FUNCTION_BLOCK FB_FieldCodecUInt32 IMPLEMENTS I_FieldCodec
VAR_INPUT
END_VAR
VAR_OUTPUT
END_VAR
VAR
    nValue : DINT;
END_VAR

METHOD CalculatePackedDataSize : HRESULT
VAR_INPUT CONSTANT
	anyFirstElem	: T_Any;
	nLength	        : UDINT;        // items to write
END_VAR
VAR_OUTPUT
    nPackedDataSize : UDINT;
END_VAR
VAR
    anyItem         : T_ANY;
    i               : UDINT;
    nValue          : UDINT;
END_VAR
anyItem := anyFirstElem;

IF nLength < 1 THEN
    nPackedDataSize := 0;
    RETURN;
END_IF

FOR i := 0  TO nLength - 1 DO
    anyItem.pValue := anyFirstElem.pValue + (i * TO_UDINT(anyFirstElem.diSize));
    MEMCPY(destAddr:= ADR(nValue), srcAddr:= anyItem.pValue, n:= TO_UDINT(anyFirstElem.diSize));
    nPackedDataSize := nPackedDataSize + F_ComputeUInt32Size(nValue);
END_FOR
END_METHOD

METHOD IsPackedRepeatedField : BOOL
VAR_INPUT
	nTag	: UDINT;
END_VAR
IsPackedRepeatedField := F_IsPackedRepeatedField(nTag);
END_METHOD


METHOD ValueReader : HRESULT
VAR_IN_OUT      
    stCtx : ST_ParseContext;
END_VAR
VAR_OUTPUT
	anyOut	: T_Any;
END_VAR

ValueReader := F_ParseRawVarint32(stCtx, nValue);
anyOut := F_ToAnyType(anyArg:= nValue);
END_METHOD

METHOD ValueWriter : HRESULT
VAR_IN_OUT
    stCtx  : ST_WriteContext;
END_VAR
VAR_INPUT
	anyIn	: ANY;
END_VAR
VAR
    nValue  : UDINT;
END_VAR

// nValue := PUDINT_TO_UDINT(anyIn.pValue);
MEMCPY(destAddr:= ADR(nValue), srcAddr:= anyIn.pValue, n:= TO_UDINT(anyIn.diSize));
ValueWriter := F_WriteUInt32(stCtx, nValue);
END_METHOD

END_FUNCTION_BLOCK

(* stored: Version 1.1.0.1
   POU FB_FieldCodecUInt32: Id {65e787ec-494b-4a47-a750-1e70e9a278a2}, SpecialFunc None
   Method CalculatePackedDataSize: Id {8b6ca985-cf9a-47d2-b259-fad382f9c60e}
   Method IsPackedRepeatedField: Id {4fbc3fd0-d99f-4835-88b1-9d66b0f4a24d}
   Method ValueReader: Id {4c83271b-1e30-4f01-9fbe-2c14057e30c1}
   Method ValueWriter: Id {f1e76788-fd58-419b-bf43-131ca6059542} *)
